FUNCTION_BLOCK RobotLadder
VAR_OUTPUT
	taskFailed : BOOL;
END_VAR
VAR
	cmd AT %Q* : TaskList; //server writes directly to this
	moveDist AT %Q* : WORD;
	
	statusReg AT %I* : UINT;
	
	rangefinderReading AT %I* : UINT;
	
	bAtHome AT %I* : BOOL;
	bAtPos1 AT %I* : BOOL;
	bAtPos2 AT %I* : BOOL;
	bMovedUp AT %I* : BOOL;
	bMovedDown AT %I* : BOOL;
	
	bMoving AT %I* : BOOL;

	timeout : TON;
	step : (IDLE, EXECUTE, FINISHED);
	done : BOOL;
END_VAR
VAR // added by the converter: edge detectors and wires of the graphical bodies
    _w1, _w2, _w3, _w4 : BOOL;
END_VAR

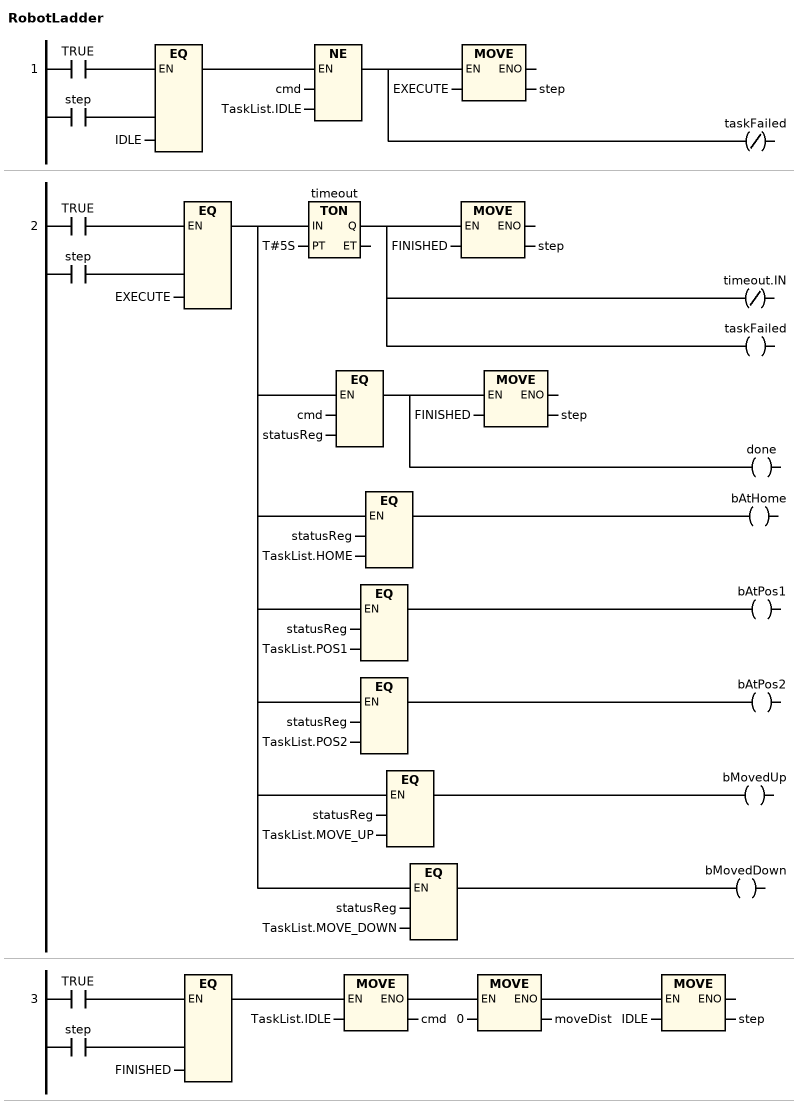
// NETWORK 1
_w1 := step = IDLE AND cmd <> TaskList.IDLE;
IF _w1 THEN step := EXECUTE; END_IF
taskFailed := NOT _w1;

// NETWORK 2
_w2 := step = EXECUTE;
timeout(IN := _w2, PT := T#5S); // TON
IF timeout.Q THEN step := FINISHED; END_IF
timeout.IN := NOT timeout.Q;
taskFailed := timeout.Q;
_w3 := _w2 AND cmd = statusReg;
IF _w3 THEN step := FINISHED; END_IF
done := _w3;
bAtHome := _w2 AND statusReg = TaskList.HOME;
bAtPos1 := _w2 AND statusReg = TaskList.POS1;
bAtPos2 := _w2 AND statusReg = TaskList.POS2;
bMovedUp := _w2 AND statusReg = TaskList.MOVE_UP;
bMovedDown := _w2 AND statusReg = TaskList.MOVE_DOWN;

// NETWORK 3
_w4 := step = FINISHED;
IF _w4 THEN cmd := TaskList.IDLE; END_IF
IF _w4 THEN moveDist := 0; END_IF
IF _w4 THEN step := IDLE; END_IF

END_FUNCTION_BLOCK

(* stored: Version 1.1.0.1, ProductVersion 3.1.4024.11
   POU RobotLadder: Id {1e189680-b8b9-4b03-8ab8-b4193f61d194}, SpecialFunc None *)
